FUNCTION_BLOCK FB_03
VAR_INPUT
END_VAR
VAR_OUTPUT
END_VAR
VAR
END_VAR

END_FUNCTION_BLOCK

(* stored: Version 1.1.0.1, ProductVersion 3.1.4024.12
   POU FB_03: Id {000c5e17-ab5b-41e0-8e75-c5b70c7a134a}, SpecialFunc None *)
